PROGRAM Initial
VAR
END_VAR

IF  GVL_System.All_Initial AND GVL_System.Manual_Mode THEN
	GVL_Vision.Data_Read_X					:=	0;
	GVL_Vision.Data_Read_Y					:=	0;
	GVL_Vision.Data_Read_R					:=	0;
	GVL_Vision.Data_Buffer_X				:=	0;
	GVL_Vision.Data_Buffer_Y				:=	0;
	GVL_Vision.Data_Buffer_R				:=	0;
	GVL_Vision.Vision_OK					:=	0;
	GVL_Vision.Data_Read_OK					:=	0;
	GVL_Vision.Data_Read_NG					:=	0;
	GVL_Vision.Target_X_Real_Position_Data	:=	0;
	GVL_Axis02.Work_Offset					:=	0;
	GVL_Main_Step.NO 						:=	0;
	GVL_Motion_Step.No						:=	0;
	GVL_Vision.Data_Check					:=	0;
	GVL_Vision.Vision_OK					:= FALSE;
	GVL_Axis04.M_Cleaning_Move := FALSE;
	GVL_Vision.Cam_Trigger := FALSE;
	GVL_Axis04.M_Mastering_Pos_Move := FALSE;
	

	// 원점 이동중/대기위치 이동중 상태 강제 해제 — 초기화 버튼으로 탈출 가능하게
	GVL_System.ALL_Home_Move_Start		:= FALSE;
	GVL_System.Axis01_Home_Move			:= FALSE;
	GVL_System.Axis02_Home_Move			:= FALSE;
	GVL_System.Axis03_Home_Move			:= FALSE;
	GVL_System.Axis04_Home_Move			:= FALSE;
	GVL_System.All_Axis_Wait_Pos_Moving	:= FALSE;
	GVL_System.Axis01_Wait_Pos_Move		:= FALSE;
	GVL_System.Axis02_Wait_Pos_Move		:= FALSE;
	GVL_System.Axis03_Wait_Pos_Move		:= FALSE;
	GVL_System.Axis04_Wait_Pos_Move		:= FALSE;
	GVL_Calibration.Calibration_Pos_Moving := FALSE;
	GVL_Calibration.Motor_Move := FALSE;

END_IF

END_PROGRAM

(* stored: Version 1.1.0.1, ProductVersion 3.1.4024.16
   POU Initial: Id {6fb955ac-b607-42dc-a361-3602f789715b}, SpecialFunc None *)
